(* CODESYS project ROBO_RECOVERED_2026-05-11T16-28-42.project

Project tree, tasks and I/O mapping:
  Device : CODESYS Control Win V3 x64, CODESYS, version 3.5.20.10
    application Application
      libraries: Standard, 3.5.18.0 (System)
      task MainTask (cyclic, interval t#20ms, priority 1) calls PLC_PRG
      program PLC_PRG [LD]
    Ethernet : Ethernet, CODESYS, version 4.2.0.0
      Modbus_TCP_Master : Modbus TCP Master, CODESYS, version 4.3.0.0
          settings: AutoReconnect = TRUE
        Modbus_TCP_Slave : Modbus TCP Slave, CODESYS, version 4.1.0.0
            settings: Unit-ID = 1; IPAddress = [192, 168, 10, 40]; Channel 0.Function Code = 2; Channel 0.Read Offset = 16#0000; Channel 0.Read Length = 9; Channel 0.Write Offset = 0; Channel 0.Write Length = 0; Channel 0.Cycle Time = 100; Channel 1.Function Code = 15; Channel 1.Read Offset = 0; Channel 1.Read Length = 0; Channel 1.Write Offset = 16#0000; Channel 1.Write Length = 15; Channel 1.Cycle Time = 100; Channel 2.Function Code = 16; Channel 2.Read Offset = 0; Channel 2.Read Length = 0; Channel 2.Write Offset = 16#0000; Channel 2.Write Length = 2; Channel 2.Cycle Time = 100
            input  LidsAtEntry : BOOL  // Channel 0.Channel 0.Bit0
            input  LidsCenterBusy : BOOL  // Channel 0.Channel 0.Bit1
            input  LidsCenterError : BOOL  // Channel 0.Channel 0.Bit2
            input  LidsAtExit : BOOL  // Channel 0.Channel 0.Bit3
            input  BasesAtEntry : BOOL  // Channel 0.Channel 0.Bit4
            input  BasesCenterBusy : BOOL  // Channel 0.Channel 0.Bit5
            input  BasesCenterError : BOOL  // Channel 0.Channel 0.Bit6
            input  BasesAtExit : BOOL  // Channel 0.Channel 0.Bit7
            input  FIO_Runing : BOOL  // Channel 0.Channel 0.Bit0
            output LidsRawConveyor : BOOL  // Channel 1.Channel 1.Bit0
            output LCProduceLids : BOOL  // Channel 1.Channel 1.Bit1
            output LCStart : BOOL  // Channel 1.Channel 1.Bit2
            output LCReset : BOOL  // Channel 1.Channel 1.Bit3
            output LCStop : BOOL  // Channel 1.Channel 1.Bit4
            output LidsExitConveyor1 : BOOL  // Channel 1.Channel 1.Bit5
            output LidsExitConveyor2 : BOOL  // Channel 1.Channel 1.Bit6
            output BasesRawConveyor : BOOL  // Channel 1.Channel 1.Bit7
            output BCProduceLids : BOOL  // Channel 1.Channel 1.Bit0
            output BCStart : BOOL  // Channel 1.Channel 1.Bit1
            output BCReset : BOOL  // Channel 1.Channel 1.Bit2
            output BCStop : BOOL  // Channel 1.Channel 1.Bit3
            output BasesExitConveyor1 : BOOL  // Channel 1.Channel 1.Bit4
            output BasesExitConveyor2 : BOOL  // Channel 1.Channel 1.Bit5
            output ExitConveyor : BOOL  // Channel 1.Channel 1.Bit6
            output LidsCounter : WORD  // Channel 2.Channel 2
            output BasesCounter : WORD  // Channel 2.Channel 2
            unmapped channels: Channel 0, Channel 1, Channel 2
*)

// Device/Application/PLC_PRG
PROGRAM PLC_PRG
VAR
	F_TRIG: ARRAY[1..4] OF F_TRIG;
	TP: ARRAY[1..2] OF TP;
	Tempo: ARRAY[1..2] OF TIME;
END_VAR
VAR // added by the converter: edge detectors and wires of the graphical bodies
    _ft1, _ft2 : F_TRIG;
END_VAR

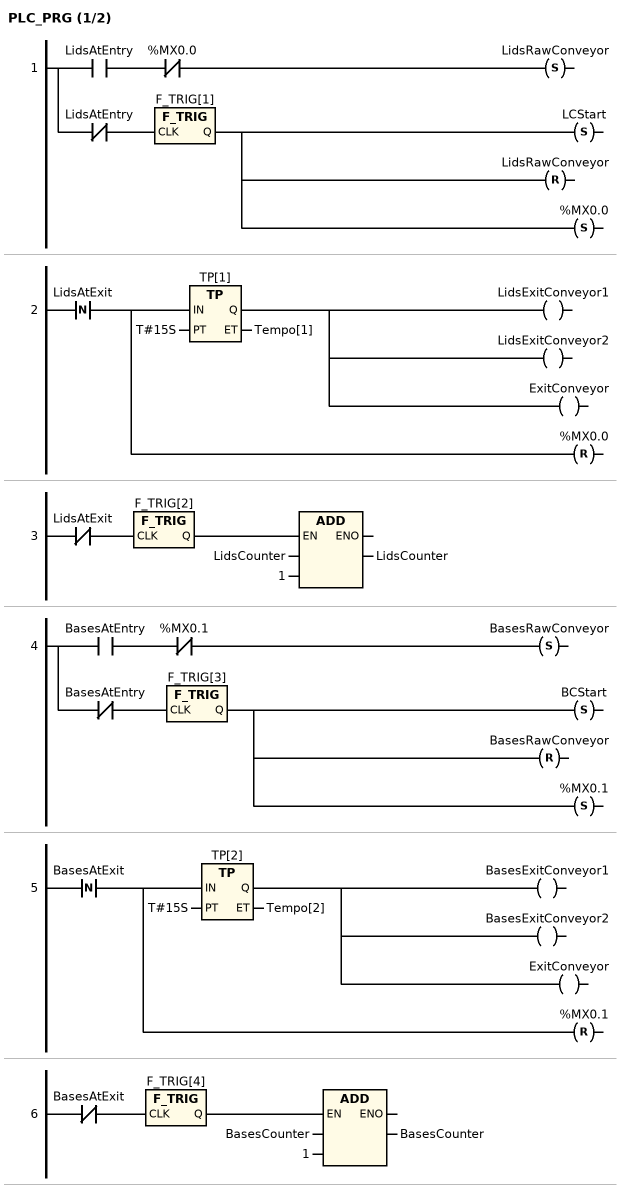
// NETWORK 1
LidsRawConveyor S= LidsAtEntry AND NOT %MX0.0;
F_TRIG[1](CLK := NOT LidsAtEntry); // F_TRIG
LCStart S= F_TRIG[1].Q;
LidsRawConveyor R= F_TRIG[1].Q;
%MX0.0 S= F_TRIG[1].Q;

// NETWORK 2
_ft1(CLK := LidsAtExit);
TP[1](IN := _ft1.Q, PT := T#15S, ET => Tempo[1]); // TP
LidsExitConveyor1 := TP[1].Q;
LidsExitConveyor2 := TP[1].Q;
ExitConveyor := TP[1].Q;
%MX0.0 R= _ft1.Q;

// NETWORK 3
F_TRIG[2](CLK := NOT LidsAtExit); // F_TRIG
IF F_TRIG[2].Q THEN LidsCounter := LidsCounter + 1; END_IF

// NETWORK 4
BasesRawConveyor S= BasesAtEntry AND NOT %MX0.1;
F_TRIG[3](CLK := NOT BasesAtEntry); // F_TRIG
BCStart S= F_TRIG[3].Q;
BasesRawConveyor R= F_TRIG[3].Q;
%MX0.1 S= F_TRIG[3].Q;

// NETWORK 5
_ft2(CLK := BasesAtExit);
TP[2](IN := _ft2.Q, PT := T#15S, ET => Tempo[2]); // TP
BasesExitConveyor1 := TP[2].Q;
BasesExitConveyor2 := TP[2].Q;
ExitConveyor := TP[2].Q;
%MX0.1 R= _ft2.Q;

// NETWORK 6
F_TRIG[4](CLK := NOT BasesAtExit); // F_TRIG
IF F_TRIG[4].Q THEN BasesCounter := BasesCounter + 1; END_IF

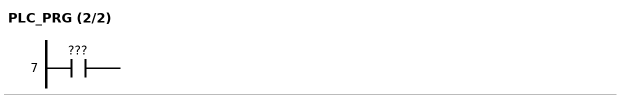
// NETWORK 7

END_PROGRAM
